PROGRAM MAIN
VAR
        test AT%MD0 : DINT;
END_VAR

test := test + 1;

END_PROGRAM

(* stored: Version 1.1.0.1, ProductVersion 3.1.4022.12
   POU MAIN: Id {626a6be7-f420-40bf-91e1-8cc14f381bec}, SpecialFunc None *)
